(* IEC 61131-3 sources: PraktykiBr/BottlePlant2/Software/Code/UserMgmt/UserCtrl, 2 files *)

(* ---- Main.st ---- *)
PROGRAM _INIT
	(* Insert code here *)
	UserCtrl.Login.Enable:=TRUE;
	UserCtrl.LoginUI.Enable:=TRUE;
	UserCtrl.UserManagerUI.Enable:=TRUE;
END_PROGRAM

PROGRAM _CYCLIC
	(* Insert code here *)
	UserCtrl.Login.MpLink:=ADR(gUserLogin);
	UserCtrl.LoginUI.MpLink:=ADR(gUserLogin);
	UserCtrl.UserManagerUI.MpLink:=ADR(gUserLogin);

	UserCtrl.LoginUI.UIConnect:=ADR(UserCtrl.UIConnect);
	UserCtrl.UserManagerUI.UIConnect:=ADR(UserCtrl.UserManagerUIConnect);
	UserCtrl.UserManagerUI.UISetup:=UserCtrl.UserManagerUISetup;

	UserCtrl.Login.UserName:=ADR(UserCtrl.UserData.UserName);
	UserCtrl.Login.Password:=ADR(UserCtrl.UserData.UserPasswd);
	gCurrentUser:=UserCtrl.Login.CurrentLevel;
	UserCtrl.Login.Logout:=gLogOutUser; // przekazanie lvl do głownego programu
	UserCtrl.UserData.UserNameStr:=WSTRING_TO_STRING(UserCtrl.Login.CurrentUser);
	UserCtrl.Login();
	UserCtrl.LoginUI();
	UserCtrl.UserManagerUI();
END_PROGRAM

PROGRAM _EXIT
	(* Insert code here *)

END_PROGRAM

(* ---- Variables.var ---- *)
VAR
	UserCtrl : UserCtrlType;
END_VAR

VAR CONSTANT

END_VAR
